TYPE Serial_StringFormat :
STRUCT
	Prefix : STRING;
	Surfix : STRING;
END_STRUCT
END_TYPE

(* stored: Version 1.1.0.1, ProductVersion 3.1.0.36
   DUT Serial_StringFormat: Id {b2a1a632-b222-4622-9cba-1dbfdeb7b2a5} *)
